// TIA Portal V16 export
// export: Created 2024-12-03T15:41:43.6094381Z, ExportSetting WithDefaults, DisplayName Totally Integrated Automation Portal, DisplayVersion V16 Update 6, DisplayName TIA Portal Version Control Interface, DisplayVersion V16 Update 2, DisplayName TIA Portal Openness, DisplayVersion V16 Update 6, DisplayName TIA Portal Teamcenter Gateway, DisplayVersion V16, DisplayName SINAMICS Startdrive Advanced, DisplayVersion V16 Update 5, DisplayName SINAMICS Startdrive G130, G150, S120, S150, SINAMICS MV, S210, DisplayVersion V16 Update 5, DisplayName SINAMICS Startdrive G110M, G120, G120C, G120D, G120P, G115D, DisplayVersion V16 Update 5, DisplayName STEP 7 Professional, DisplayVersion V16 Update 6, DisplayName STEP 7 Safety, DisplayVersion V16, DisplayName WinCC Advanced / Unified PC, DisplayVersion V16 Update 6
FUNCTION_BLOCK "Multiple_click_FB"   // FB115, SCL
{ S7_Optimized_Access := 'TRUE' }
VERSION : 0.1
// stored: AutoNumber true, IsIECCheckEnabled false, IsRetainMemResEnabled false, MemoryReserve 100, SetENOAutomatically false, UDAEnableTagReadback false
   VAR_INPUT
      I_Signal : "SmartBooldt";
      I_Clicks : UInt;
   END_VAR
   VAR_OUTPUT
      O_SignalClick : Bool;
   END_VAR
   VAR
      iddle : TON_TIME;
      counts { S7_SetPoint := 'True'} : UInt;
   END_VAR
BEGIN
   REGION TIMINGS

       #O_SignalClick := FALSE;

       #iddle(IN:=true,
              PT:=t#700ms);

       IF #iddle.Q THEN
           #counts := 0;
       END_IF;

       IF #I_Signal.LE THEN
           RESET_TIMER(#iddle);
       END_IF;

       IF #I_Signal.LE AND NOT #iddle.Q THEN
           #counts += 1;
       END_IF;

       IF #counts >= #I_Clicks THEN
           #counts := 0;
           #O_SignalClick := true;
       END_IF;

   END_REGION
END_FUNCTION_BLOCK
